// TIA Portal project "下轴装配_V15.1" (V15.1)

(* hardware
DEVICE "S7-1200 station_1"  S7-1200 Station
   slot 0: "Rack_0"  S7-1200 Rack  Rack  V1.0
   slot 1: "A170648_14 CPU  1214C"  CPU 1214C DC/DC/DC  6ES7 214-1AG40-0XB0  V4.2
   slot 2: "DI 16/DQ 16x24VDC_1"  6ES7 223-1BL32-0XB0  V2.0
   slot 3: "AQ 1x12BIT_1"  AQ1 signal board  6ES7 232-4HA30-0XB0  V1.0
   slot 3: "AI 4x13BIT_1"  SM 1231 AI4  6ES7 231-4HD30-0XB0  V1.0
*)

// ===== PLC "A170648_14 CPU  1214C"  CPU 1214C DC/DC/DC =====

VAR_GLOBAL   // PLC tag table "默认变量表"
   "启动" AT %I0.0 : Bool;
   "不" AT %I0.1 : Bool;
   "复位" AT %I0.2 : Bool;
   "急停" AT %I0.3 : Bool;
   "阻尼左" AT %I0.4 : Bool;
   "阻尼右" AT %I0.5 : Bool;
   "阻尼" AT %I0.6 : Bool;
   "toolCheck3" AT %I0.7 : Bool;
   "色标笔" AT %I1.0 : Bool;
   "toolCheck5" AT %I1.1 : Bool;
   "拧紧枪确认" AT %I1.2 : Bool;
   "不合格" AT %I1.3 : Bool;
   "合格" AT %I1.4 : Bool;
   "toolCheck9" AT %I1.5 : Bool;
   "toolCheck10" AT %I2.0 : Bool;
   "toolCheck11" AT %I2.1 : Bool;
   "toolCheck12" AT %I2.2 : Bool;
   "toolCheck13" AT %I2.3 : Bool;
   "toolCheck14" AT %I2.4 : Bool;
   "toolCheck15" AT %I2.5 : Bool;
   "噪音检测退位" AT %I2.6 : Bool;
   "噪音检测进位" AT %I2.7 : Bool;
   "Tag_18" AT %IW64 : Int;
   "噪音检测进" AT %Q0.0 : Bool;
   "噪音检测退" AT %Q0.1 : Bool;
   "噪音检测进(1)" AT %Q0.2 : Bool;
   "噪音检测退(1)" AT %Q0.3 : Bool;
   "车速" AT %Q0.4 : Bool;
   "点火" AT %Q0.5 : Bool;
   "转速" AT %Q0.6 : Bool;
   "备用(14)" AT %Q0.7 : Bool;
   "合格指示灯" AT %Q1.0 : Bool;
   "不合格指示灯" AT %Q1.1 : Bool;
   "防护门上升" AT %Q2.0 : Bool;
   "防护门下降" AT %Q2.1 : Bool;
   "绿" AT %Q2.2 : Bool;
   "黄" AT %Q2.3 : Bool;
   "红" AT %Q2.4 : Bool;
   "蜂鸣器" AT %Q2.5 : Bool;
   "备用(17)" AT %Q2.6 : Bool;
   "备用(18)" AT %Q2.7 : Bool;
   "检具选取(1)" AT %Q20.0 : Bool;
   "检具选取(2)" AT %Q20.1 : Bool;
   "检具选取(3)" AT %Q20.2 : Bool;
   "检具选取(4)" AT %Q20.3 : Bool;
   "检具选取(5)" AT %Q20.4 : Bool;
   "检具选取(6)" AT %Q20.5 : Bool;
   "检具选取(7)" AT %Q20.6 : Bool;
   "检具拾取(8)" AT %Q20.7 : Bool;
   "检具选取(9)" AT %Q21.0 : Bool;
   "检具选取(10)" AT %Q21.1 : Bool;
   "检具选取(11)" AT %Q21.2 : Bool;
   "检具选取(12)" AT %Q21.3 : Bool;
   "检具选取(13)" AT %Q21.4 : Bool;
   "检具选取(14)" AT %Q21.5 : Bool;
   "检具选取(15)" AT %Q21.6 : Bool;
   "检具选取(16)" AT %Q21.7 : Bool;
   "Tag_17" AT %QW80 : Int;
   "Tag_21" AT %Q3.2 : Bool;
   "程序停止" AT %M100.0 : Bool;
   "复位完成" AT %M100.1 : Bool;
   "Clock_1Hz" AT %M0.5 : Bool;
   "AlwaysFALSE" AT %M1.3 : Bool;
   "Clock_Byte" AT %MB0 : Byte;
   "Clock_10Hz" AT %M0.0 : Bool;
   "Clock_5Hz" AT %M0.1 : Bool;
   "Clock_2.5Hz" AT %M0.2 : Bool;
   "Clock_2Hz" AT %M0.3 : Bool;
   "Clock_1.25Hz" AT %M0.4 : Bool;
   "Clock_0.625Hz" AT %M0.6 : Bool;
   "Clock_0.5Hz" AT %M0.7 : Bool;
   "System_Byte" AT %MB1 : Byte;
   "FirstScan" AT %M1.0 : Bool;
   "DiagStatusUpdate" AT %M1.1 : Bool;
   "AlwaysTRUE" AT %M1.2 : Bool;
   "拾取步_9" AT %M202.0 : Bool;
   "拾取步_10" AT %M202.1 : Bool;
   "拾取步_11" AT %M202.2 : Bool;
   "拾取步_12" AT %M202.3 : Bool;
   "拾取步_13" AT %M202.4 : Bool;
   "拾取步_14" AT %M202.5 : Bool;
   "拾取步_15" AT %M202.6 : Bool;
   "拾取步_16" AT %M202.7 : Bool;
   "拾取步_1" AT %M203.0 : Bool;
   "拾取步_2" AT %M203.1 : Bool;
   "拾取步_3" AT %M203.2 : Bool;
   "拾取步_4" AT %M203.3 : Bool;
   "拾取步_5" AT %M203.4 : Bool;
   "拾取步_6" AT %M203.5 : Bool;
   "拾取步_7" AT %M203.6 : Bool;
   "拾取步_8" AT %M203.7 : Bool;
   "拾取步_17" AT %M300.0 : Bool;
   "拾取报错" AT %M400.0 : Bool;
   "检具选取" AT %MW100 : Word;
   "拾取步" AT %MW202 : Word;
   "Tag_1" AT %M306.0 : Bool;
   "Tag_2" AT %M306.1 : Bool;
   "Tag_3" AT %M306.2 : Bool;
   "Tag_4" AT %M306.3 : Bool;
   "Tag_5" AT %M306.4 : Bool;
   "Tag_6" AT %M306.5 : Bool;
   "Tag_7" AT %M306.6 : Bool;
   "Tag_8" AT %M306.7 : Bool;
   "Tag_9" AT %M307.0 : Bool;
   "Tag_10" AT %M307.1 : Bool;
   "Tag_11" AT %M307.2 : Bool;
   "Tag_12" AT %M307.3 : Bool;
   "Tag_13" AT %M307.4 : Bool;
   "Tag_14" AT %M307.5 : Bool;
   "Tag_15" AT %M307.6 : Bool;
   "Tag_16" AT %M307.7 : Bool;
   "拾取开启" AT %MW306 : Word;
   "Tag_19" AT %MD200 : Real;
   "Tag_20" AT %MD204 : Real;
   "磁粉离合器校准" AT %M160.0 : Bool;
   "Tag_22" AT %M300.1 : Bool;
   "Tag_23" AT %M300.2 : Bool;
   "Tag_24" AT %M300.3 : Bool;
   "Tag_25" AT %M303.0 : Bool;
   "Tag_26" AT %M303.1 : Bool;
   "Tag_27" AT %M303.2 : Bool;
   "Tag_28" AT %M303.3 : Bool;
   "Tag_29" AT %IW12 : Int;
   "Tag_30" AT %IW112 : Word;
END_VAR

DATA_BLOCK "SERVER"   // DB1
{ S7_Optimized_Access := 'FALSE' }
VERSION : 0.1
   VAR
      设备状态 : Int := 0;
      产品型号 : Int := 0;
      错误代码 : Int := 0;
      生产结果 : Int := 0;
      设备编号 : Int := 0;
      产品标识 : Int;
      下轴安装螺栓数 : Int;
      转动圈数 : Int;
      转动阻尼设置 : Int;
      传感器参数 : Array[0..2] of Real;
   END_VAR
BEGIN
   // 传感器参数[2] : scl采集
END_DATA_BLOCK

DATA_BLOCK "MB_TCON"   // DB2
{ S7_Optimized_Access := 'FALSE' }
VERSION : 0.1
   VAR
      MB_TCON : TCON_IP_v4;
   END_VAR
BEGIN
   MB_TCON.InterfaceId := 64;
   MB_TCON.ID := 1;
   MB_TCON.LocalPort := 502;
   MB_TCON.RemoteAddress.ADDR[1] := 0;
   MB_TCON.RemoteAddress.ADDR[2] := 0;
   MB_TCON.RemoteAddress.ADDR[3] := 0;
   MB_TCON.RemoteAddress.ADDR[4] := 0;
END_DATA_BLOCK

DATA_BLOCK "RESET_DB"   // DB3
{ S7_Optimized_Access := 'TRUE' }
VERSION : 0.1
// stored: InstanceOfName RESET
"RESET"
BEGIN
END_DATA_BLOCK

DATA_BLOCK "ALARM_DB"   // DB4
{ S7_Optimized_Access := 'TRUE' }
VERSION : 0.1
// stored: InstanceOfName ALARM
"ALARM"
BEGIN
END_DATA_BLOCK

DATA_BLOCK "AUTO_DB"   // DB10
{ S7_Optimized_Access := 'TRUE' }
VERSION : 0.1
// stored: InstanceOfName AUTO
"AUTO"
BEGIN
END_DATA_BLOCK

DATA_BLOCK "SERVER_Rapid"   // DB15
{ S7_Optimized_Access := 'TRUE' }
VERSION : 0.1
   VAR
      传感器参数1 : Real;
   END_VAR
BEGIN
END_DATA_BLOCK

DATA_BLOCK "采集_DB"   // DB16
{ S7_Optimized_Access := 'TRUE' }
VERSION : 0.1
// stored: InstanceOfName 采集
"采集"
BEGIN
END_DATA_BLOCK

DATA_BLOCK "车速1"   // DB20
{ S7_Optimized_Access := 'TRUE' }
VERSION : 0.1
   VAR
      speed1 : Int;
   END_VAR
BEGIN
END_DATA_BLOCK

// folder: System blocks/Program resources

DATA_BLOCK "IEC_Timer_0_DB"   // DB5
{ S7_Optimized_Access := 'TRUE' }
AUTHOR : Simatic
FAMILY : IEC
NAME : IEC_TMR
VERSION : 1.0
// stored: InstanceOfName IEC_TIMER
"IEC_TIMER"
BEGIN
END_DATA_BLOCK

DATA_BLOCK "IEC_Timer_0_DB_3"   // DB12
{ S7_Optimized_Access := 'TRUE' }
AUTHOR : Simatic
FAMILY : IEC
NAME : IEC_TMR
VERSION : 1.0
// stored: InstanceOfName IEC_TIMER
"IEC_TIMER"
BEGIN
END_DATA_BLOCK

// folder: (top level)

DATA_BLOCK "轴_1"   // DB6, Motion_DB
{ S7_Optimized_Access := 'TRUE' }
AUTHOR : SIMATIC
FAMILY : BasicMC
NAME : TO_PosAx
VERSION : 6.0
// stored: InstanceOfName TO_PositioningAxis
"TO_PositioningAxis"
BEGIN
   // Axis.SelectedChannel2EnumCU = %Q0.5
   // Axis.DirectionOutputEnabledCU = TRUE
   // Axis.OnlinePtoIndexCU = 2
   // Axis.OnlinePtoModeCUEnumValue = PTO（脉冲 A 和方向 B）
   // Axis.OnlinePtoModeCU = 16#0000_0002
   // Axis.SelectedChannel1EnumCU = %Q0.4
   // Pulse.MinDeltaDeltaFrequencyCU = 0.004
   // Pulse.MaxDeltaDeltaFrequencyCU = 1.0E+10
   // Pulse.MinDeltaFrequencyCU = 0.005
   // Pulse.MaxDeltaFrequencyCU = 9.5E+9
   // Pulse.MinFrequencyCU = 1.0
   // Pulse.MaxFrequencyCU = 30000.0
   // Pulse.OutputSourceCU = 16#0000_0000
   // Axis.SelectPTO = 2
   // Axis.LengthUnit.LastDistance = -1
END_DATA_BLOCK

DATA_BLOCK "轴_2"   // DB7, Motion_DB
{ S7_Optimized_Access := 'TRUE' }
AUTHOR : SIMATIC
FAMILY : BasicMC
NAME : TO_PosAx
VERSION : 6.0
// stored: InstanceOfName TO_PositioningAxis
"TO_PositioningAxis"
BEGIN
   // Axis.OnlinePtoModeCUEnumValue = PTO（脉冲 A 和方向 B）
   // Axis.OnlinePtoModeCU = 16#0000_0002
   // Axis.SelectedChannel1EnumCU = %Q0.6
   // Pulse.MinDeltaDeltaFrequencyCU = 0.004
   // Pulse.MaxDeltaDeltaFrequencyCU = 1.0E+10
   // Pulse.MinDeltaFrequencyCU = 0.005
   // Pulse.MaxDeltaFrequencyCU = 9.5E+9
   // Pulse.MinFrequencyCU = 1.0
   // Pulse.MaxFrequencyCU = 30000.0
   // Pulse.OutputSourceCU = 16#0000_0000
   // Axis.SelectPTO = 3
   // Axis.OnlinePtoIndexCU = 3
   // Axis.LengthUnit.LastDistance = -1
END_DATA_BLOCK

FUNCTION_BLOCK "ALARM"   // FB1, LAD
{ S7_Optimized_Access := 'TRUE' }
VERSION : 0.1
   VAR
      "Error-ID" : Word;
      TEmp : Array[0..3] of Bool;
      IEC_Timer_0_Instance : TON_TIME;
      IEC_Timer_0_Instance_1 : TON_TIME;
      IEC_Timer_0_Instance_2 : TON_TIME;
      IEC_Timer_0_Instance_3 : TON_TIME;
      IEC_Timer_0_Instance_4 : TON_TIME;
      IEC_Timer_0_Instance_5 : TON_TIME;
      IEC_Timer_0_Instance_6 : TON_TIME;
      IEC_Timer_0_Instance_7 : TON_TIME;
      IEC_Timer_0_Instance_8 : TON_TIME;
      IEC_Timer_0_Instance_9 : TON_TIME;
      IEC_Timer_0_Instance_10 : TON_TIME;
      IEC_Timer_0_Instance_11 : TON_TIME;
      IEC_Timer_0_Instance_12 : TON_TIME;
      IEC_Timer_0_Instance_13 : TON_TIME;
      IEC_Timer_0_Instance_14 : TON_TIME;
      "STEP" : Int;
      IEC_Timer_0_Instance_15 : TON_TIME;
      IEC_Timer_0_Instance_16 : TON_TIME;
   END_VAR
BEGIN

REGION Network 1
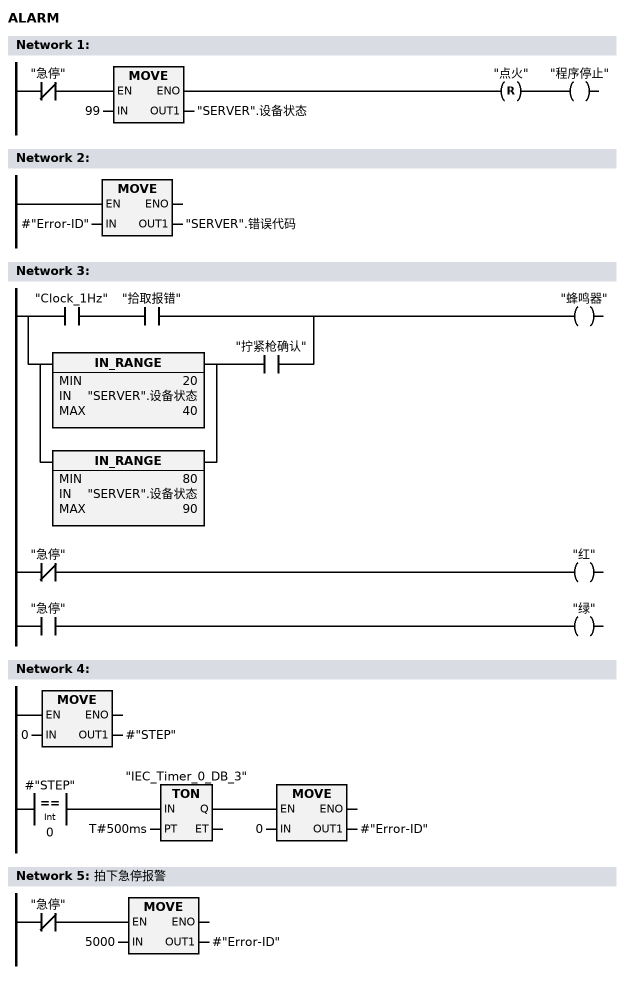
   RUNG wire#powerrail
      I_Contact( "急停" )
      Move(in := 99, out1 => "SERVER".设备状态)
      R_Coil( "点火" )
      Coil( "程序停止" )
   END_RUNG
   // the same network as SCL:
   IF NOT "急停" THEN
       "SERVER".设备状态 := 99;
       "点火" := FALSE;
   END_IF;
   "程序停止" := NOT "急停";
END_REGION

REGION Network 2
   RUNG wire#powerrail
      Move(in := #"Error-ID", out1 => "SERVER".错误代码)
   END_RUNG
   // the same network as SCL:
   "SERVER".错误代码 := #"Error-ID";
END_REGION

REGION Network 3
   RUNG wire#powerrail
      Contact( "Clock_1Hz" )
      Contact( "拾取报错" )
      wire#w1
      Coil( "蜂鸣器" )
   END_RUNG
   RUNG wire#powerrail
      { S7_Templates := "SrcType := Int" } InRange(min := 20, in := "SERVER".设备状态, max := 40)
      wire#w2
      Contact( "拧紧枪确认" )
   END_RUNG wire#w1
   RUNG wire#powerrail
      { S7_Templates := "SrcType := Int" } InRange(min := 80, in := "SERVER".设备状态, max := 90)
   END_RUNG wire#w2
   RUNG wire#powerrail
      I_Contact( "急停" )
      Coil( "红" )
   END_RUNG
   RUNG wire#powerrail
      Contact( "急停" )
      Coil( "绿" )
   END_RUNG
   // the same network as SCL:
   "蜂鸣器" := ("Clock_1Hz" AND "拾取报错") OR ((((20 <= "SERVER".设备状态) AND ("SERVER".设备状态 <= 40)) OR ((80 <= "SERVER".设备状态) AND ("SERVER".设备状态 <= 90))) AND "拧紧枪确认");
   "红" := NOT "急停";
   "绿" := "急停";
END_REGION

REGION Network 4
   #"STEP" := 0;
   "IEC_Timer_0_DB_3".TON(IN := #"STEP" = 0, PT := T#500ms);
   IF "IEC_Timer_0_DB_3".Q THEN #"Error-ID" := 0; END_IF;
END_REGION

REGION Network 5: 拍下急停报警
   RUNG wire#powerrail
      I_Contact( "急停" )
      Move(in := 5000, out1 => #"Error-ID")
   END_RUNG
   // the same network as SCL:
   IF NOT "急停" THEN #"Error-ID" := 5000; END_IF;
END_REGION

REGION Network 6: 安全门打开报警
END_REGION

REGION Network 7: 工件未在位启动报警
END_REGION

REGION Network 8: 气源未开报警
END_REGION

REGION Network 9: 工装移栽前进未到位报警
END_REGION

REGION Network 10: 工装移栽未后退报警
END_REGION

REGION Network 11: 防护门未上升报警
END_REGION

REGION Network 12: 防护门为下降报警
END_REGION

REGION Network 13: 1#固定气缸未锁紧报警
END_REGION

REGION Network 14: 1#固定气缸未退回报警
END_REGION

REGION Network 15: 1#机械手未上升报警
END_REGION

REGION Network 16: 1#机械手未下降报警
END_REGION

REGION Network 17: 1#气爪未夹紧到位报警
END_REGION

REGION Network 18: 1#气爪未松开报警
END_REGION

REGION Network 19: 2#机械手未固定锁紧报警
END_REGION

REGION Network 20: 2#固定气缸未退回报警
END_REGION

REGION Network 21: 2#机械手未上升报警
END_REGION

REGION Network 22: 2#机械手未下降报警
END_REGION

REGION Network 23: 2#气爪未夹紧报警
END_REGION

REGION Network 24: 2#气爪未松开报警
END_REGION

REGION Network 25: 激光打码报警
END_REGION
END_FUNCTION_BLOCK

FUNCTION_BLOCK "RESET"   // FB2, LAD
{ S7_Optimized_Access := 'TRUE' }
VERSION : 0.1
   VAR_INPUT
      Stop : Bool;
      Start : Bool;
   END_VAR
   VAR_OUTPUT
      Down : Bool;
   END_VAR
   VAR
      "Step" : Int;
      MC_Reset_Instance : MC_Reset;
      MC_Reset_Instance_1 : MC_Reset;
      IEC_Timer_0_Instance : TON_TIME;
   END_VAR
   VAR_TEMP   // added for the SCL form of the ladder/FBD networks
      _w1 : Bool;
   END_VAR
BEGIN

REGION Network 1
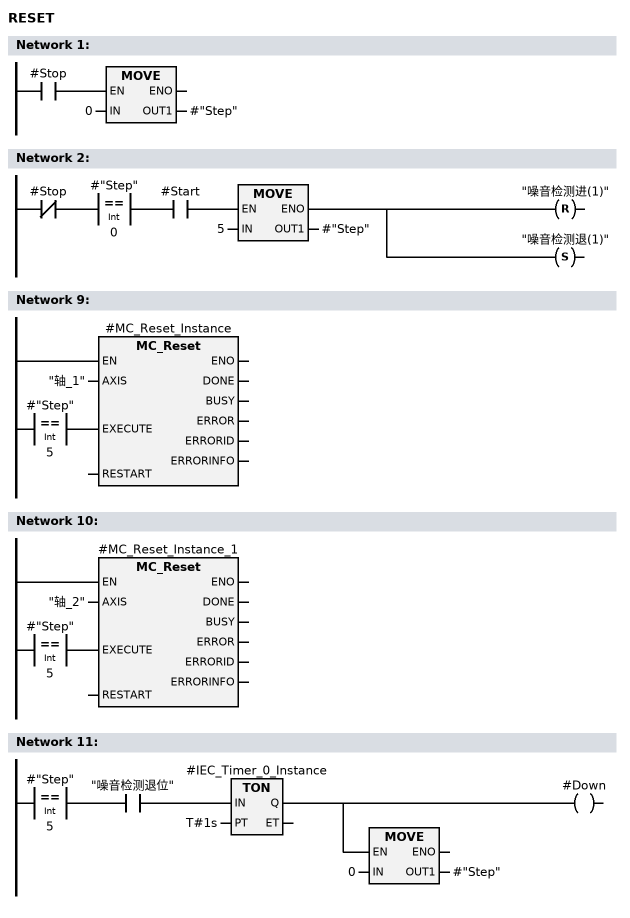
   RUNG wire#powerrail
      Contact( #Stop )
      Move(in := 0, out1 => #"Step")
   END_RUNG
   // the same network as SCL:
   IF #Stop THEN #"Step" := 0; END_IF;
END_REGION

REGION Network 2
   RUNG wire#powerrail
      I_Contact( #Stop )
      { S7_Templates := "SrcType := Int" } EQ_Contact(in1 := #"Step", in2 := 0)
      Contact( #Start )
      Move(in := 5, out1 => #"Step")
      wire#w1
      R_Coil( "噪音检测进(1)" )
   END_RUNG
   RUNG wire#w1
      S_Coil( "噪音检测退(1)" )
   END_RUNG
   // the same network as SCL:
   #_w1 := NOT #Stop AND (#"Step" = 0) AND #Start;
   IF #_w1 THEN
       #"Step" := 5;
       "噪音检测进(1)" := FALSE;
       "噪音检测退(1)" := TRUE;
   END_IF;
END_REGION

REGION Network 7: 1#气爪松开
END_REGION

REGION Network 8: 2#气爪松开
END_REGION

REGION Network 9
   #MC_Reset_Instance(Axis := "轴_1", Execute := #"Step" = 5);   // MC_Reset
END_REGION

REGION Network 10
   #MC_Reset_Instance_1(Axis := "轴_2", Execute := #"Step" = 5);   // MC_Reset
END_REGION

REGION Network 11
   #IEC_Timer_0_Instance(IN := (#"Step" = 5) AND "噪音检测退位", PT := T#1s);   // TON
   #Down := #IEC_Timer_0_Instance.Q;
   IF #IEC_Timer_0_Instance.Q THEN #"Step" := 0; END_IF;
END_REGION
END_FUNCTION_BLOCK

FUNCTION_BLOCK "AUTO"   // FB3, LAD
{ S7_Optimized_Access := 'TRUE' }
VERSION : 0.1
   VAR
      IEC_Timer_0_Instance : TON_TIME;
      IEC_Timer_0_Instance_1 : TON_TIME;
      IEC_Timer_0_Instance_2 : TON_TIME;
   END_VAR
   VAR_TEMP   // added for the SCL form of the ladder/FBD networks
      _w1 : Bool;
      _w2 : Bool;
   END_VAR
BEGIN

REGION Network 1
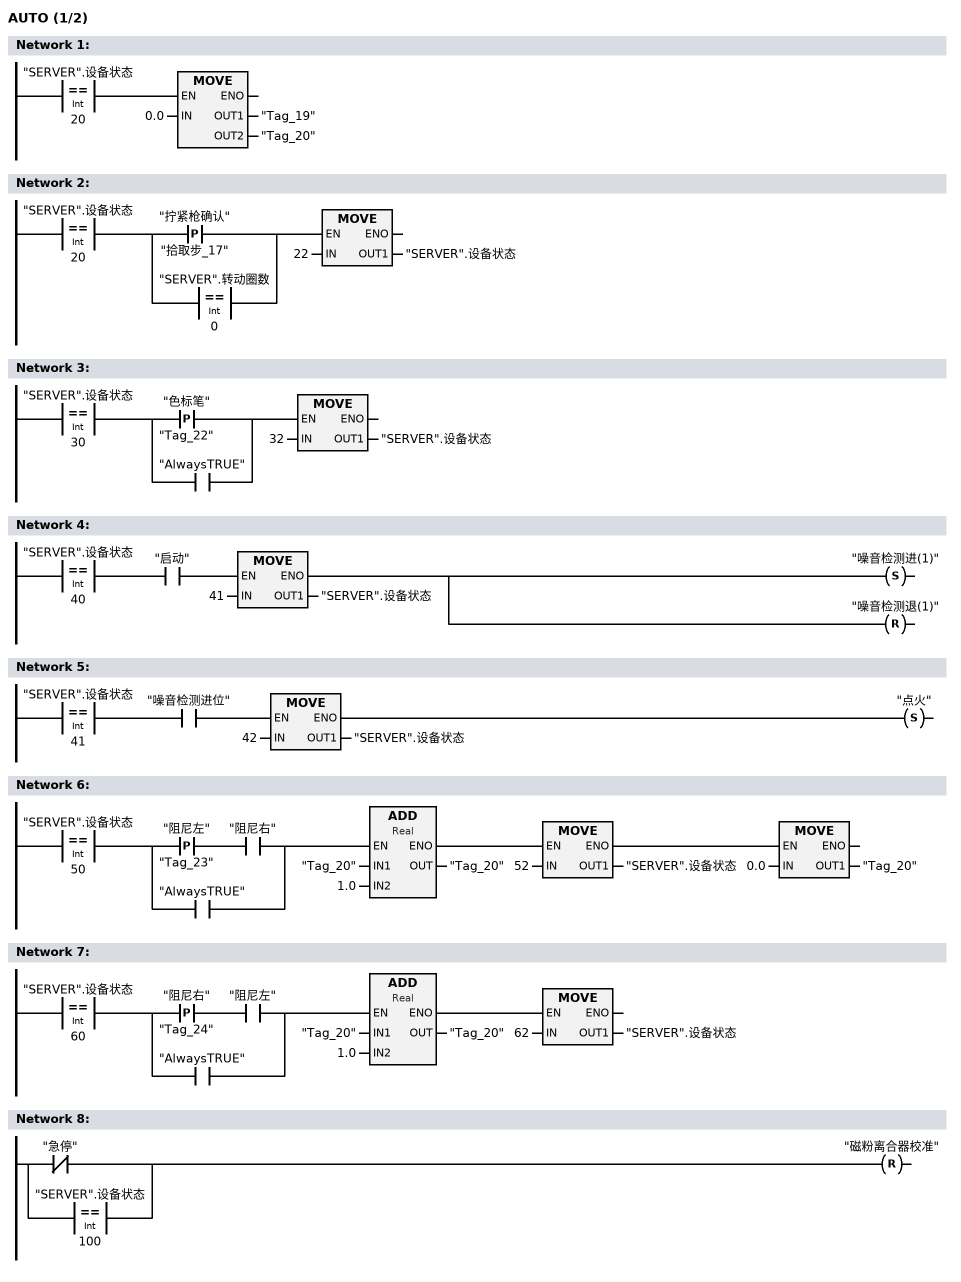
   RUNG wire#powerrail
      { S7_Templates := "SrcType := Int" } EQ_Contact(in1 := "SERVER".设备状态, in2 := 20)
      Move(in := 0.0, out1 => "Tag_19", out2 => "Tag_20")
   END_RUNG
   // the same network as SCL:
   IF "SERVER".设备状态 = 20 THEN
       "Tag_19" := 0.0;
       "Tag_20" := 0.0;
   END_IF;
END_REGION

REGION Network 2
   RUNG wire#powerrail
      { S7_Templates := "SrcType := Int" } EQ_Contact(in1 := "SERVER".设备状态, in2 := 20)
      wire#w1
      P_Contact(operand := "拧紧枪确认", bit := "拾取步_17")
      wire#w2
      Move(in := 22, out1 => "SERVER".设备状态)
   END_RUNG
   RUNG wire#w1
      { S7_Templates := "SrcType := Int" } EQ_Contact(in1 := "SERVER".转动圈数, in2 := 0)
   END_RUNG wire#w2
   // the same network as SCL:
   #_w1 := ("SERVER".设备状态 = 20) AND "拧紧枪确认" AND NOT "拾取步_17";   // rising edge of "拧紧枪确认"
   "拾取步_17" := "拧紧枪确认";
   IF #_w1 OR (("SERVER".设备状态 = 20) AND ("SERVER".转动圈数 = 0)) THEN "SERVER".设备状态 := 22; END_IF;
END_REGION

REGION Network 3
   RUNG wire#powerrail
      { S7_Templates := "SrcType := Int" } EQ_Contact(in1 := "SERVER".设备状态, in2 := 30)
      wire#w1
      P_Contact(operand := "色标笔", bit := "Tag_22")
      wire#w2
      Move(in := 32, out1 => "SERVER".设备状态)
   END_RUNG
   RUNG wire#w1
      Contact( "AlwaysTRUE" )
   END_RUNG wire#w2
   // the same network as SCL:
   #_w1 := ("SERVER".设备状态 = 30) AND "色标笔" AND NOT "Tag_22";   // rising edge of "色标笔"
   "Tag_22" := "色标笔";
   IF #_w1 OR (("SERVER".设备状态 = 30) AND "AlwaysTRUE") THEN "SERVER".设备状态 := 32; END_IF;
END_REGION

REGION Network 4
   RUNG wire#powerrail
      { S7_Templates := "SrcType := Int" } EQ_Contact(in1 := "SERVER".设备状态, in2 := 40)
      Contact( "启动" )
      Move(in := 41, out1 => "SERVER".设备状态)
      wire#w1
      S_Coil( "噪音检测进(1)" )
   END_RUNG
   RUNG wire#w1
      R_Coil( "噪音检测退(1)" )
   END_RUNG
   // the same network as SCL:
   #_w1 := ("SERVER".设备状态 = 40) AND "启动";
   IF #_w1 THEN
       "SERVER".设备状态 := 41;
       "噪音检测进(1)" := TRUE;
       "噪音检测退(1)" := FALSE;
   END_IF;
END_REGION

REGION Network 5
   RUNG wire#powerrail
      { S7_Templates := "SrcType := Int" } EQ_Contact(in1 := "SERVER".设备状态, in2 := 41)
      Contact( "噪音检测进位" )
      Move(in := 42, out1 => "SERVER".设备状态)
      S_Coil( "点火" )
   END_RUNG
   // the same network as SCL:
   #_w1 := ("SERVER".设备状态 = 41) AND "噪音检测进位";
   IF #_w1 THEN
       "SERVER".设备状态 := 42;
       "点火" := TRUE;
   END_IF;
END_REGION

REGION Network 6
   RUNG wire#powerrail
      { S7_Templates := "SrcType := Int" } EQ_Contact(in1 := "SERVER".设备状态, in2 := 50)
      wire#w1
      P_Contact(operand := "阻尼左", bit := "Tag_23")
      Contact( "阻尼右" )
      wire#w2
      { S7_Templates := "SrcType := Real" } Add(in1 := "Tag_20", in2 := 1.0, out => "Tag_20")
      Move(in := 52, out1 => "SERVER".设备状态)
      Move(in := 0.0, out1 => "Tag_20")
   END_RUNG
   RUNG wire#w1
      Contact( "AlwaysTRUE" )
   END_RUNG wire#w2
   // the same network as SCL:
   #_w1 := ("SERVER".设备状态 = 50) AND "阻尼左" AND NOT "Tag_23";   // rising edge of "阻尼左"
   "Tag_23" := "阻尼左";
   IF (#_w1 AND "阻尼右") OR (("SERVER".设备状态 = 50) AND "AlwaysTRUE") THEN "Tag_20" := "Tag_20" + 1.0; END_IF;
   #_w2 := (#_w1 AND "阻尼右") OR (("SERVER".设备状态 = 50) AND "AlwaysTRUE");
   IF #_w2 THEN
       "SERVER".设备状态 := 52;
       "Tag_20" := 0.0;
   END_IF;
END_REGION

REGION Network 7
   RUNG wire#powerrail
      { S7_Templates := "SrcType := Int" } EQ_Contact(in1 := "SERVER".设备状态, in2 := 60)
      wire#w1
      P_Contact(operand := "阻尼右", bit := "Tag_24")
      Contact( "阻尼左" )
      wire#w2
      { S7_Templates := "SrcType := Real" } Add(in1 := "Tag_20", in2 := 1.0, out => "Tag_20")
      Move(in := 62, out1 => "SERVER".设备状态)
   END_RUNG
   RUNG wire#w1
      Contact( "AlwaysTRUE" )
   END_RUNG wire#w2
   // the same network as SCL:
   #_w1 := ("SERVER".设备状态 = 60) AND "阻尼右" AND NOT "Tag_24";   // rising edge of "阻尼右"
   "Tag_24" := "阻尼右";
   IF (#_w1 AND "阻尼左") OR (("SERVER".设备状态 = 60) AND "AlwaysTRUE") THEN
       "Tag_20" := "Tag_20" + 1.0;
       "SERVER".设备状态 := 62;
   END_IF;
END_REGION

REGION Network 8
   RUNG wire#powerrail
      I_Contact( "急停" )
      wire#w1
      R_Coil( "磁粉离合器校准" )
   END_RUNG
   RUNG wire#powerrail
      { S7_Templates := "SrcType := Int" } EQ_Contact(in1 := "SERVER".设备状态, in2 := 100)
   END_RUNG wire#w1
   // the same network as SCL:
   IF NOT "急停" OR ("SERVER".设备状态 = 100) THEN "磁粉离合器校准" := FALSE; END_IF;
END_REGION

REGION Network 9
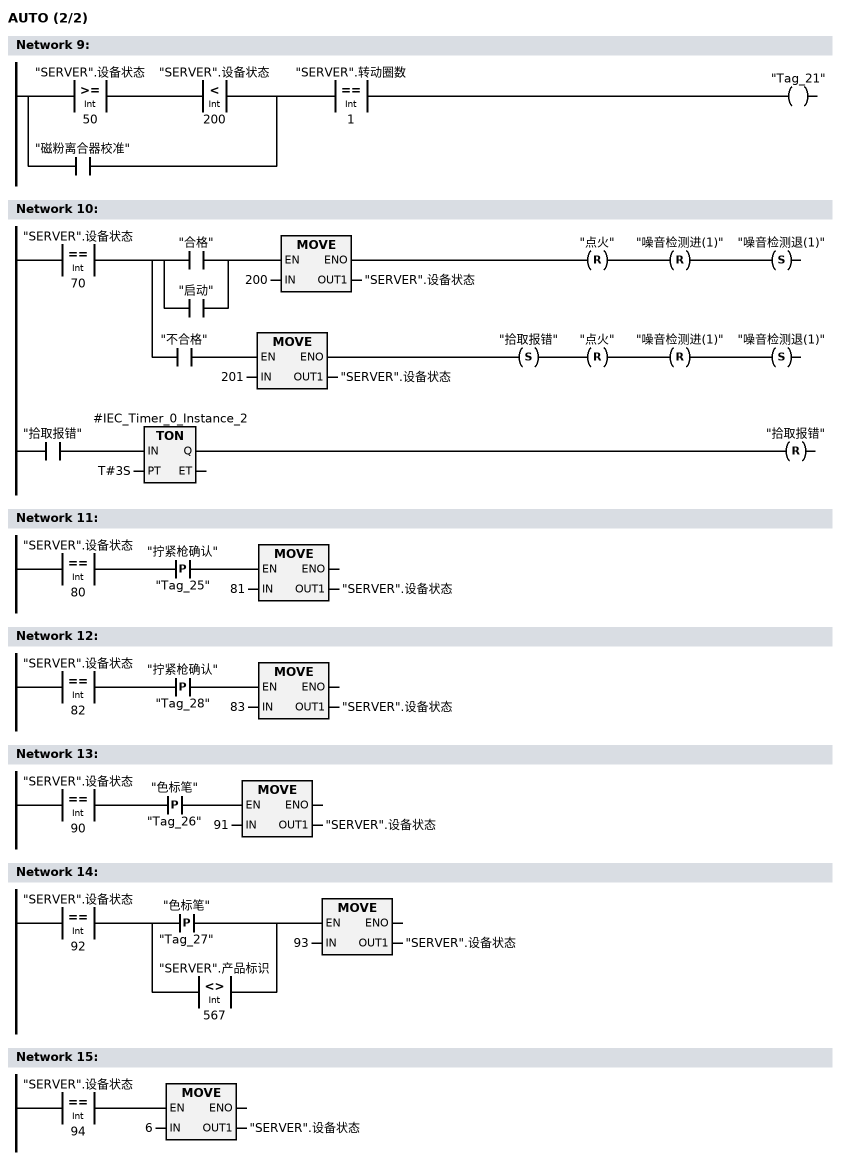
   RUNG wire#powerrail
      { S7_Templates := "SrcType := Int" } GE_Contact(in1 := "SERVER".设备状态, in2 := 50)
      { S7_Templates := "SrcType := Int" } LT_Contact(in1 := "SERVER".设备状态, in2 := 200)
      wire#w1
      { S7_Templates := "SrcType := Int" } EQ_Contact(in1 := "SERVER".转动圈数, in2 := 1)
      Coil( "Tag_21" )
   END_RUNG
   RUNG wire#powerrail
      Contact( "磁粉离合器校准" )
   END_RUNG wire#w1
   // the same network as SCL:
   "Tag_21" := ((("SERVER".设备状态 >= 50) AND ("SERVER".设备状态 < 200)) OR "磁粉离合器校准") AND ("SERVER".转动圈数 = 1);
END_REGION

REGION Network 10
   #_w1 := "SERVER".设备状态 = 70;
   IF #_w1 AND ("合格" OR "启动") THEN
       "SERVER".设备状态 := 200;
       "点火" := FALSE;
       "噪音检测进(1)" := FALSE;
       "噪音检测退(1)" := TRUE;
   END_IF;
   IF #_w1 AND "不合格" THEN
       "SERVER".设备状态 := 201;
       "拾取报错" := TRUE;
       "点火" := FALSE;
       "噪音检测进(1)" := FALSE;
       "噪音检测退(1)" := TRUE;
   END_IF;
   #IEC_Timer_0_Instance_2(IN := "拾取报错", PT := T#3S);   // TON
   IF #IEC_Timer_0_Instance_2.Q THEN "拾取报错" := FALSE; END_IF;
END_REGION

REGION Network 11
   RUNG wire#powerrail
      { S7_Templates := "SrcType := Int" } EQ_Contact(in1 := "SERVER".设备状态, in2 := 80)
      P_Contact(operand := "拧紧枪确认", bit := "Tag_25")
      Move(in := 81, out1 => "SERVER".设备状态)
   END_RUNG
   // the same network as SCL:
   #_w1 := ("SERVER".设备状态 = 80) AND "拧紧枪确认" AND NOT "Tag_25";   // rising edge of "拧紧枪确认"
   "Tag_25" := "拧紧枪确认";
   IF #_w1 THEN "SERVER".设备状态 := 81; END_IF;
END_REGION

REGION Network 12
   RUNG wire#powerrail
      { S7_Templates := "SrcType := Int" } EQ_Contact(in1 := "SERVER".设备状态, in2 := 82)
      P_Contact(operand := "拧紧枪确认", bit := "Tag_28")
      Move(in := 83, out1 => "SERVER".设备状态)
   END_RUNG
   // the same network as SCL:
   #_w1 := ("SERVER".设备状态 = 82) AND "拧紧枪确认" AND NOT "Tag_28";   // rising edge of "拧紧枪确认"
   "Tag_28" := "拧紧枪确认";
   IF #_w1 THEN "SERVER".设备状态 := 83; END_IF;
END_REGION

REGION Network 13
   RUNG wire#powerrail
      { S7_Templates := "SrcType := Int" } EQ_Contact(in1 := "SERVER".设备状态, in2 := 90)
      P_Contact(operand := "色标笔", bit := "Tag_26")
      Move(in := 91, out1 => "SERVER".设备状态)
   END_RUNG
   // the same network as SCL:
   #_w1 := ("SERVER".设备状态 = 90) AND "色标笔" AND NOT "Tag_26";   // rising edge of "色标笔"
   "Tag_26" := "色标笔";
   IF #_w1 THEN "SERVER".设备状态 := 91; END_IF;
END_REGION

REGION Network 14
   RUNG wire#powerrail
      { S7_Templates := "SrcType := Int" } EQ_Contact(in1 := "SERVER".设备状态, in2 := 92)
      wire#w1
      P_Contact(operand := "色标笔", bit := "Tag_27")
      wire#w2
      Move(in := 93, out1 => "SERVER".设备状态)
   END_RUNG
   RUNG wire#w1
      { S7_Templates := "SrcType := Int" } NE_Contact(in1 := "SERVER".产品标识, in2 := 567)
   END_RUNG wire#w2
   // the same network as SCL:
   #_w1 := ("SERVER".设备状态 = 92) AND "色标笔" AND NOT "Tag_27";   // rising edge of "色标笔"
   "Tag_27" := "色标笔";
   IF #_w1 OR (("SERVER".设备状态 = 92) AND ("SERVER".产品标识 <> 567)) THEN "SERVER".设备状态 := 93; END_IF;
END_REGION

REGION Network 15
   RUNG wire#powerrail
      { S7_Templates := "SrcType := Int" } EQ_Contact(in1 := "SERVER".设备状态, in2 := 94)
      Move(in := 6, out1 => "SERVER".设备状态)
   END_RUNG
   // the same network as SCL:
   IF "SERVER".设备状态 = 94 THEN "SERVER".设备状态 := 6; END_IF;
END_REGION
END_FUNCTION_BLOCK

FUNCTION_BLOCK "采集"   // FB4, SCL
{ S7_Optimized_Access := 'TRUE' }
VERSION : 0.1
   VAR_INPUT
      采集值 : Real;
      设备上限 : Real;
      设备下限 : Real;
      清零 : Bool;
   END_VAR
   VAR_OUTPUT
      工程值 : Real;
   END_VAR
   VAR
      零点漂移 : Real;
   END_VAR
BEGIN
   #工程值 := #采集值 * (#设备上限 - #设备下限) /( 27648*2) + #设备下限-#零点漂移;
   IF #清零 THEN
       // Statement section IF
       #零点漂移:=#工程值 ;

   END_IF;
END_FUNCTION_BLOCK

FUNCTION "拾取" : Void   // FC1, LAD
{ S7_Optimized_Access := 'TRUE' }
VERSION : 0.1
   VAR_INPUT
      拾取0 : Bool;
      拾取1 : Bool;
      拾取2 : Bool;
      拾取3 : Bool;
      拾取4 : Bool;
      拾取5 : Bool;
      拾取6 : Bool;
      拾取7 : Bool;
      拾取8 : Bool;
      拾取9 : Bool;
      拾取10 : Bool;
      拾取11 : Bool;
      拾取12 : Bool;
      拾取13 : Bool;
      拾取14 : Bool;
      拾取15 : Bool;
   END_VAR
   VAR_TEMP
      temp : Word;
   END_VAR
   VAR_TEMP   // added for the SCL form of the ladder/FBD networks
      _w1 : Bool;
   END_VAR
BEGIN

REGION Network 1
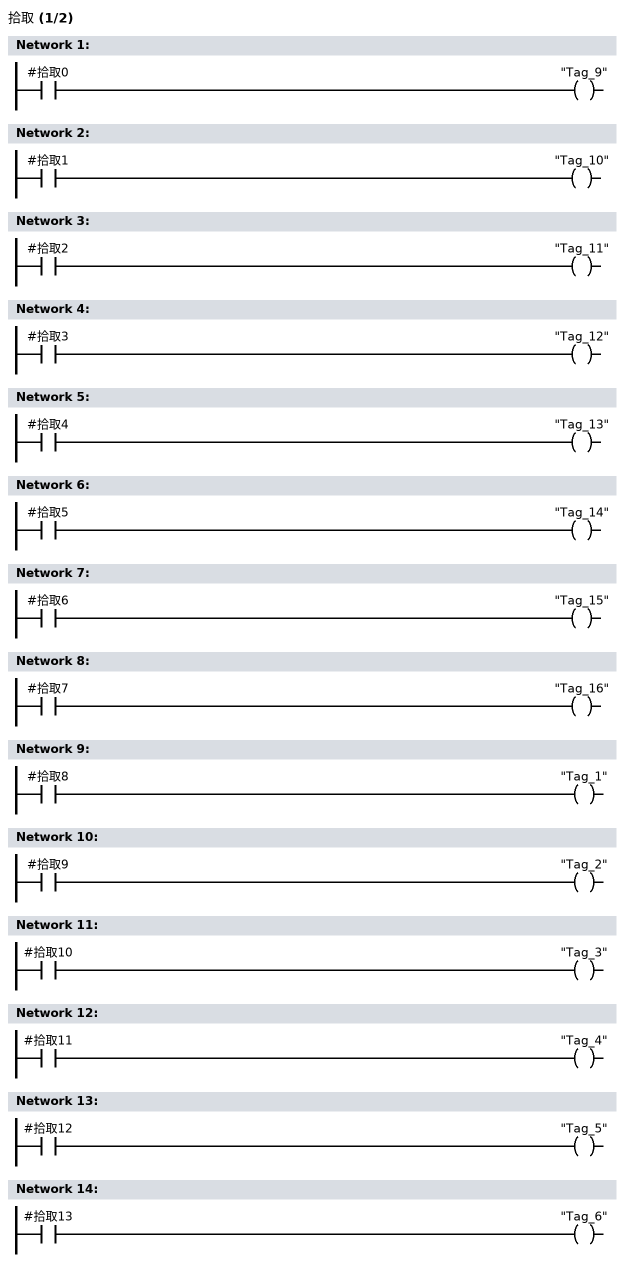
   RUNG wire#powerrail
      Contact( #拾取0 )
      Coil( "Tag_9" )
   END_RUNG
   // the same network as SCL:
   "Tag_9" := #拾取0;
END_REGION

REGION Network 2
   RUNG wire#powerrail
      Contact( #拾取1 )
      Coil( "Tag_10" )
   END_RUNG
   // the same network as SCL:
   "Tag_10" := #拾取1;
END_REGION

REGION Network 3
   RUNG wire#powerrail
      Contact( #拾取2 )
      Coil( "Tag_11" )
   END_RUNG
   // the same network as SCL:
   "Tag_11" := #拾取2;
END_REGION

REGION Network 4
   RUNG wire#powerrail
      Contact( #拾取3 )
      Coil( "Tag_12" )
   END_RUNG
   // the same network as SCL:
   "Tag_12" := #拾取3;
END_REGION

REGION Network 5
   RUNG wire#powerrail
      Contact( #拾取4 )
      Coil( "Tag_13" )
   END_RUNG
   // the same network as SCL:
   "Tag_13" := #拾取4;
END_REGION

REGION Network 6
   RUNG wire#powerrail
      Contact( #拾取5 )
      Coil( "Tag_14" )
   END_RUNG
   // the same network as SCL:
   "Tag_14" := #拾取5;
END_REGION

REGION Network 7
   RUNG wire#powerrail
      Contact( #拾取6 )
      Coil( "Tag_15" )
   END_RUNG
   // the same network as SCL:
   "Tag_15" := #拾取6;
END_REGION

REGION Network 8
   RUNG wire#powerrail
      Contact( #拾取7 )
      Coil( "Tag_16" )
   END_RUNG
   // the same network as SCL:
   "Tag_16" := #拾取7;
END_REGION

REGION Network 9
   RUNG wire#powerrail
      Contact( #拾取8 )
      Coil( "Tag_1" )
   END_RUNG
   // the same network as SCL:
   "Tag_1" := #拾取8;
END_REGION

REGION Network 10
   RUNG wire#powerrail
      Contact( #拾取9 )
      Coil( "Tag_2" )
   END_RUNG
   // the same network as SCL:
   "Tag_2" := #拾取9;
END_REGION

REGION Network 11
   RUNG wire#powerrail
      Contact( #拾取10 )
      Coil( "Tag_3" )
   END_RUNG
   // the same network as SCL:
   "Tag_3" := #拾取10;
END_REGION

REGION Network 12
   RUNG wire#powerrail
      Contact( #拾取11 )
      Coil( "Tag_4" )
   END_RUNG
   // the same network as SCL:
   "Tag_4" := #拾取11;
END_REGION

REGION Network 13
   RUNG wire#powerrail
      Contact( #拾取12 )
      Coil( "Tag_5" )
   END_RUNG
   // the same network as SCL:
   "Tag_5" := #拾取12;
END_REGION

REGION Network 14
   RUNG wire#powerrail
      Contact( #拾取13 )
      Coil( "Tag_6" )
   END_RUNG
   // the same network as SCL:
   "Tag_6" := #拾取13;
END_REGION

REGION Network 15
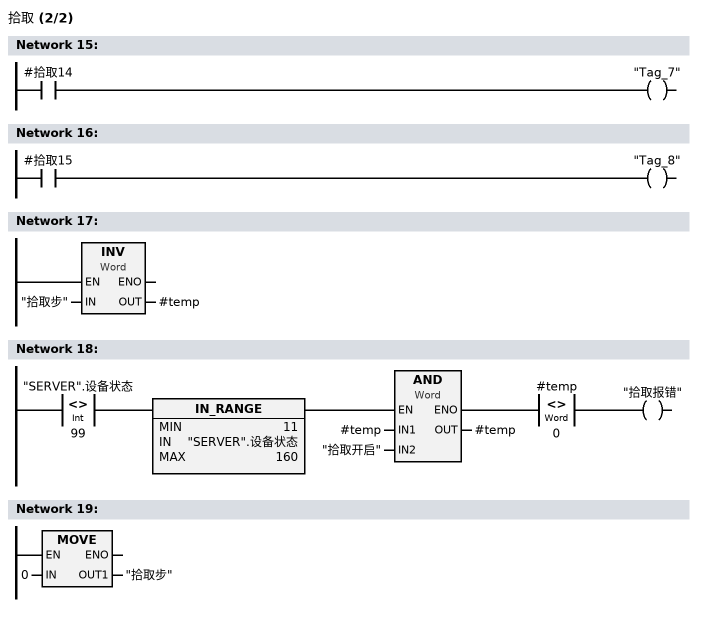
   RUNG wire#powerrail
      Contact( #拾取14 )
      Coil( "Tag_7" )
   END_RUNG
   // the same network as SCL:
   "Tag_7" := #拾取14;
END_REGION

REGION Network 16
   RUNG wire#powerrail
      Contact( #拾取15 )
      Coil( "Tag_8" )
   END_RUNG
   // the same network as SCL:
   "Tag_8" := #拾取15;
END_REGION

REGION Network 17
   RUNG wire#powerrail
      { S7_Templates := "SrcType := Word" } Inv(in := "拾取步", out => #temp)
   END_RUNG
   // the same network as SCL:
   #temp := NOT "拾取步";
END_REGION

REGION Network 18
   RUNG wire#powerrail
      { S7_Templates := "SrcType := Int" } NE_Contact(in1 := "SERVER".设备状态, in2 := 99)
      { S7_Templates := "SrcType := Int" } InRange(min := 11, in := "SERVER".设备状态, max := 160)
      { S7_Templates := "SrcType := Word" } And(in1 := #temp, in2 := "拾取开启", out => #temp)
      { S7_Templates := "SrcType := Word" } NE_Contact(in1 := #temp, in2 := 0)
      Coil( "拾取报错" )
   END_RUNG
   // the same network as SCL:
   #_w1 := ("SERVER".设备状态 <> 99) AND (11 <= "SERVER".设备状态) AND ("SERVER".设备状态 <= 160);
   IF #_w1 THEN #temp := #temp AND "拾取开启"; END_IF;
   "拾取报错" := #_w1 AND (#temp <> 0);
END_REGION

REGION Network 19
   RUNG wire#powerrail
      Move(in := 0, out1 => "拾取步")
   END_RUNG
   // the same network as SCL:
   "拾取步" := 0;
END_REGION
END_FUNCTION

FUNCTION "int to real" : Void   // FC3, LAD
{ S7_Optimized_Access := 'TRUE' }
VERSION : 0.1
   VAR_INPUT
      vaule : Int;
      maxOut : Real;
   END_VAR
   VAR_OUTPUT
      out : Real;
   END_VAR
   VAR_TEMP
      real_i : Real;
      real_q : Real;
      minOut : Real;
   END_VAR
BEGIN

REGION Network 1
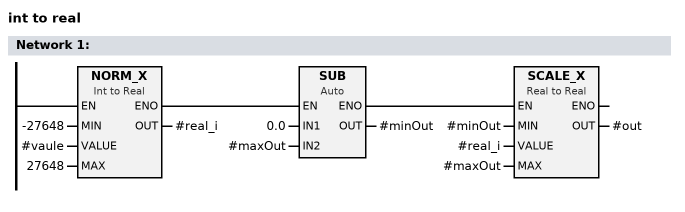
   RUNG wire#powerrail
      { S7_Templates := "[SrcType := Int, DestType := Real]" } Normalize(min := -27648, value := #vaule, max := 27648, out => #real_i)
      Sub(in1 := 0.0, in2 := #maxOut, out => #minOut)
      { S7_Templates := "[SrcType := Real, DestType := Real]" } Scale(min := #minOut, value := #real_i, max := #maxOut, out => #out)
   END_RUNG
   // the same network as SCL:
   #real_i := NORM_X(MIN := -27648, VALUE := #vaule, MAX := 27648);
   #minOut := 0.0 - #maxOut;
   #out := SCALE_X(MIN := #minOut, VALUE := #real_i, MAX := #maxOut);
END_REGION
END_FUNCTION

ORGANIZATION_BLOCK "Main"   // OB1, LAD, ProgramCycle
TITLE = "Main Program Sweep (Cycle)"
{ S7_Optimized_Access := 'TRUE' }
VERSION : 0.1
   VAR_INPUT
      Initial_Call : Bool;   // Initial call of this OB
      Remanence : Bool;   // =True, if remanent data are available
   END_VAR
   VAR_TEMP   // added for the SCL form of the ladder/FBD networks
      _w1 : Bool;
   END_VAR
BEGIN

REGION Network 1
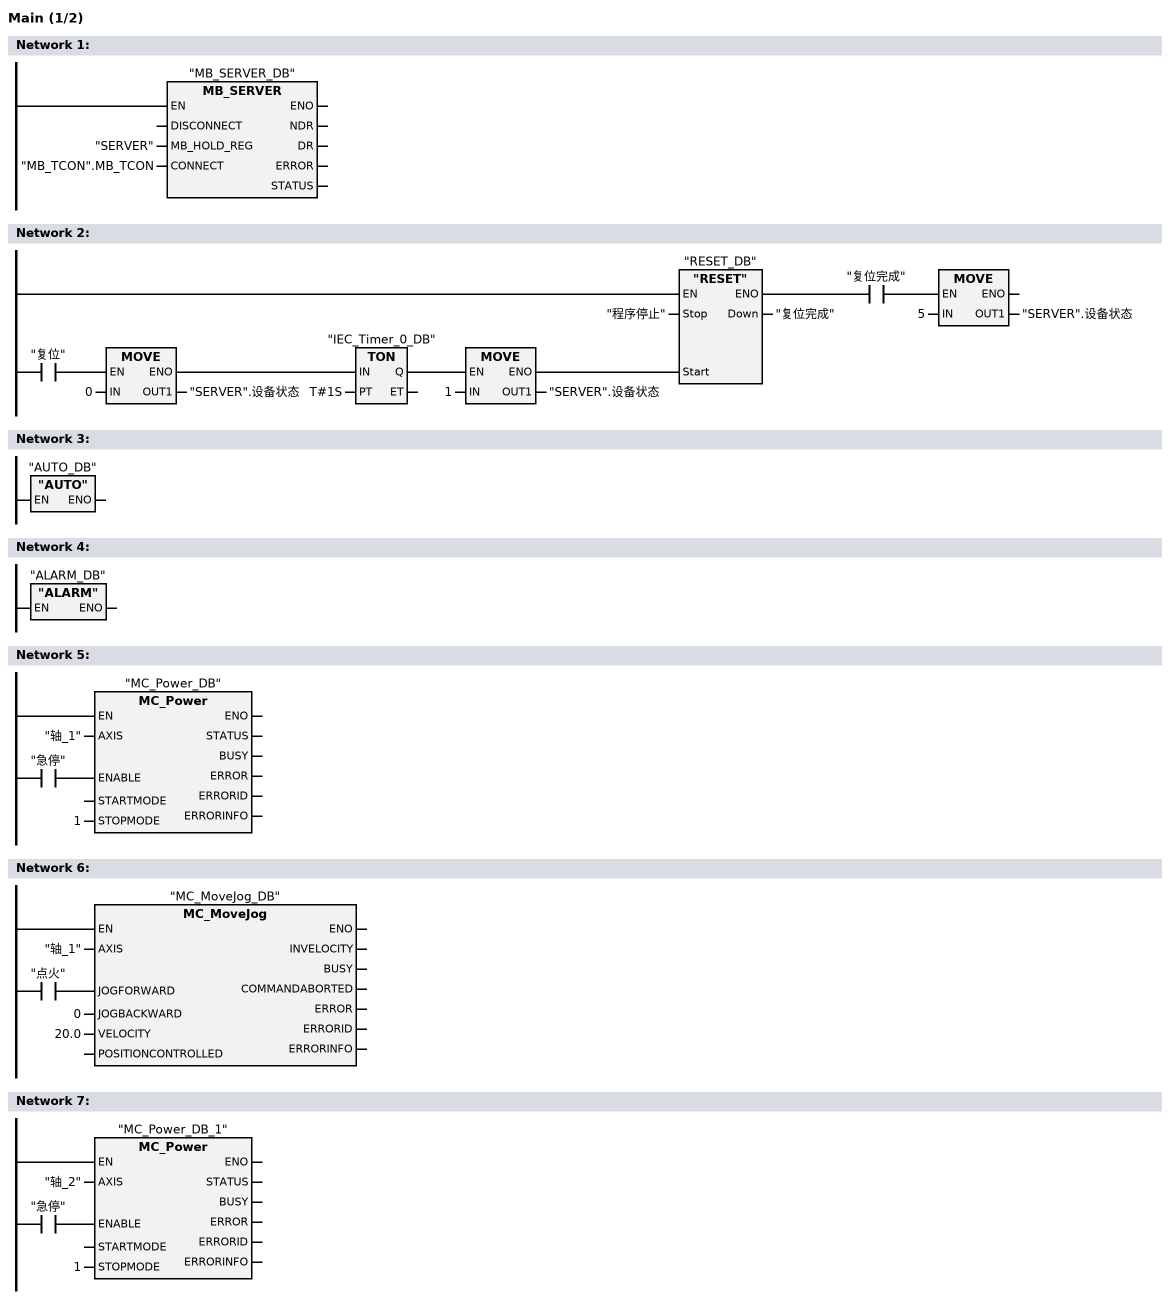
   "MB_SERVER_DB"(MB_HOLD_REG := "SERVER", CONNECT := "MB_TCON".MB_TCON);   // MB_SERVER
END_REGION

REGION Network 2
   IF "复位" THEN "SERVER".设备状态 := 0; END_IF;
   "IEC_Timer_0_DB".TON(IN := "复位", PT := T#1S);
   IF "IEC_Timer_0_DB".Q THEN "SERVER".设备状态 := 1; END_IF;
   "RESET_DB"(Stop := "程序停止", Start := "IEC_Timer_0_DB".Q, Down => "复位完成", ENO => #_w1);   // "RESET"
   IF #_w1 AND "复位完成" THEN "SERVER".设备状态 := 5; END_IF;
END_REGION

REGION Network 3
   RUNG wire#powerrail
      "AUTO_DB"()
   END_RUNG
   // the same network as SCL:
   "AUTO_DB"();   // "AUTO"
END_REGION

REGION Network 4
   RUNG wire#powerrail
      "ALARM_DB"()
   END_RUNG
   // the same network as SCL:
   "ALARM_DB"();   // "ALARM"
END_REGION

REGION Network 5
   "MC_Power_DB"(Axis := "轴_1", Enable := "急停", StopMode := 1);   // MC_Power
END_REGION

REGION Network 6
   "MC_MoveJog_DB"(Axis := "轴_1", JogForward := "点火", JogBackward := 0, Velocity := 20.0);   // MC_MoveJog
END_REGION

REGION Network 7
   "MC_Power_DB_1"(Axis := "轴_2", Enable := "急停", StopMode := 1);   // MC_Power
END_REGION

REGION Network 8
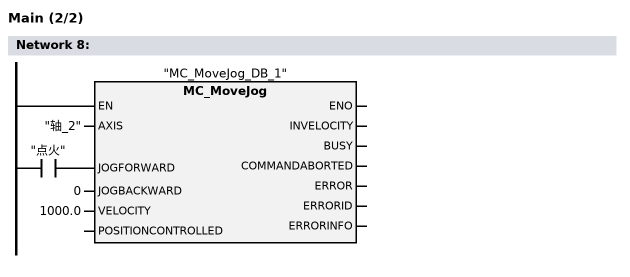
   "MC_MoveJog_DB_1"(Axis := "轴_2", JogForward := "点火", JogBackward := 0, Velocity := 1000.0);   // MC_MoveJog
END_REGION
END_ORGANIZATION_BLOCK

ORGANIZATION_BLOCK "Cyclic interrupt_10ms"   // OB30, LAD, CyclicInterrupt
{ S7_Optimized_Access := 'TRUE' }
VERSION : 0.1
   VAR_INPUT
      Initial_Call : Bool;   // Initial call of this OB
      Event_Count : Int;   // Events discarded
   END_VAR
   VAR_TEMP
      done : Bool;
      done_1 : Bool;
      busy : Bool;
      direction : Bool;
      speed : Real;
      temp2 : Int;
      temp1 : Real;
      temp3 : Real;
      torque : Real;
      Tag_18R : Int;
   END_VAR
BEGIN

REGION Network 1
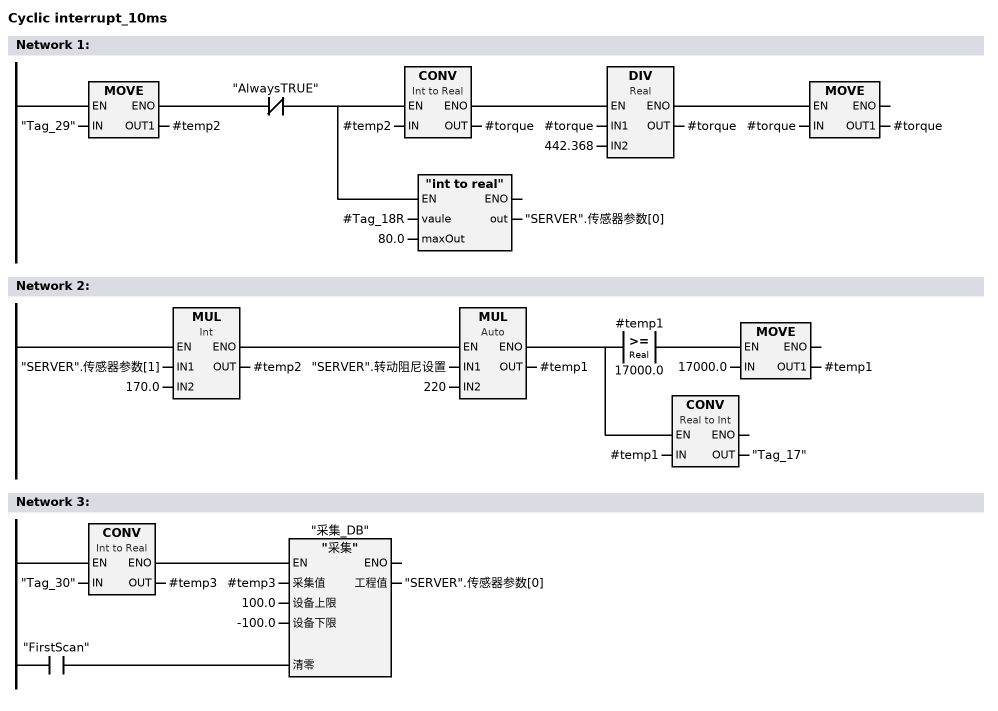
   RUNG wire#powerrail
      Move(in := "Tag_29", out1 => #temp2)
      I_Contact( "AlwaysTRUE" )
      wire#w1
      { S7_Templates := "[SrcType := Int, DestType := Real]" } Convert(in := #temp2, out => #torque)
      { S7_Templates := "SrcType := Real" } Div(in1 := #torque, in2 := 442.368, out => #torque)
      Move(in := #torque, out1 => #torque)
   END_RUNG
   RUNG wire#w1
      "int to real"(vaule := #Tag_18R, maxOut := 80.0, out => "SERVER".传感器参数[0])
   END_RUNG
   // the same network as SCL:
   #temp2 := "Tag_29";
   IF NOT "AlwaysTRUE" THEN
       #torque := INT_TO_REAL(#temp2);
       #torque := #torque / 442.368;
       #torque := #torque;
       "int to real"(vaule := #Tag_18R, maxOut := 80.0, out => "SERVER".传感器参数[0]);
   END_IF;
END_REGION

REGION Network 2
   RUNG wire#powerrail
      { S7_Templates := "SrcType := Int" } Mul(in1 := "SERVER".传感器参数[1], in2 := 170.0, out => #temp2)
      Mul(in1 := "SERVER".转动阻尼设置, in2 := 220, out => #temp1)
      wire#w1
      { S7_Templates := "SrcType := Real" } GE_Contact(in1 := #temp1, in2 := 17000.0)
      Move(in := 17000.0, out1 => #temp1)
   END_RUNG
   RUNG wire#w1
      { S7_Templates := "[SrcType := Real, DestType := Int]" } Convert(in := #temp1, out => "Tag_17")
   END_RUNG
   // the same network as SCL:
   #temp2 := "SERVER".传感器参数[1] * 170.0;
   #temp1 := "SERVER".转动阻尼设置 * 220;
   IF #temp1 >= 17000.0 THEN #temp1 := 17000.0; END_IF;
   "Tag_17" := REAL_TO_INT(#temp1);
END_REGION

REGION Network 3
   RUNG wire#powerrail
      { S7_Templates := "[SrcType := Int, DestType := Real]" } Convert(in := "Tag_30", out => #temp3)
      "采集_DB"(清零 := wire#w1, 采集值 := #temp3, 设备上限 := 100.0, 设备下限 := -100.0, 工程值 => "SERVER".传感器参数[0])
   END_RUNG
   RUNG wire#powerrail
      Contact( "FirstScan" )
   END_RUNG wire#w1
   // the same network as SCL:
   #temp3 := INT_TO_REAL("Tag_30");
   "采集_DB"(采集值 := #temp3, 设备上限 := 100.0, 设备下限 := -100.0, 清零 := "FirstScan", 工程值 => "SERVER".传感器参数[0]);   // "采集"
END_REGION
END_ORGANIZATION_BLOCK